TYPE "LBP_typeAxisX"
TITLE = Axis interface / Interfaz de eje / Achsschnittstelle
// User data type for blocks LBP_Axis1 [DB31] .. LBP_Axis31 [DB61] / Tipo de dato de usuario para bloques LBP_Axis1 [DB31] .. LBP_Axis31 [DB61] / Anwender-Datentyp für Bausteine LBP_Axis1 [DB31] .. LBP_Axis31 [DB61]
// stored: IsFailsafeCompliant false
   STRUCT
      A_FD_OR : Byte;   // Vorschub-Override / Feedrate override / Corrección de avance
      A_DriveEnable : Bool;   // Antriebstest-Bewegung aktivieren / Drive test movement enable / Habilitar movimiento test accionamiento
      A_AckFixedStop : Bool;   // Quittieren Festanschlag erreicht / Acknowledge fixed stop reached / Confirmar tope fijo alcanzado
      A_SensorFixedStop : Bool;   // Sensor Festanschlag / Sensor fixed stop / Sensor tope fijo
      A_ASpDisable : Bool;   // Achse/Spindel deaktivieren / Axis/spindle disable / Deshabilitar eje/cabezal
      A_Follow_upMode : Bool;   // Nachlaufbetrieb / Follow-up mode / Modo de seguimiento
      A_PosMeas1 : Bool;   // Positionsmesssystem 1 / Position measuring system 1 / Sistema de medida de posición 1
      A_PosMeas2 : Bool;   // Positionsmesssystem 2 / Position measuring system 2 / Sistema de medida de posición 2
      A_ORactive : Bool;   // Override aktiv / Override active / Corrección activa
      A_SWCam : Bool;   // SW Nocken-Aktivierung / SW cam activation / Activación de levas de SW
      A_ContrEnable : Bool;   // Steuerung aktivieren / Controller enable / Habilitar controlador
      A_DelDTGSpReset : Bool;   // Restweg löschen/Spindel-Reset / Delete distance to go/Spindle-Reset / Borrar trayecto residual/reset de cabezal
      A_Clamp : Bool;   // Spannen läuft / Clamping in progress / Amarre en curso
      A_RefVal1 : Bool;   // Referenzpunktwert 1 / Reference point value 1 / Valor de punto de referencia 1
      A_RefVal2 : Bool;   // Referenzpunktwert 2 / Reference point value 2 / Valor de punto de referencia 2
      A_RefVal3 : Bool;   // Referenzpunktwert 3 / Reference point value 3 / Valor de punto de referencia 3
      A_RefVal4 : Bool;   // Referenzpunktwert 4 / Reference point value 4 / Valor de punto de referencia 4
      A_ExtZO : Bool;   // Externe ZO importieren / Import external ZO / Importar ZO externo
      A_EnabTravFixedStop : Bool;   // Verfahren zu Festanschlag aktivieren / Enable travel to fixed stop / Activar desplazamiento a tope fijo
      A_FixedFD1 : Bool;   // Festen Vorschub 1 aktivieren / Activate fixed feedrate 1 / Activar avance fijo 1
      A_FixedFD2 : Bool;   // Festen Vorschub 2 aktivieren / Activate fixed feedrate 2 / Activar avance fijo 2
      A_FixedFD3 : Bool;   // Festen Vorschub 3 aktivieren / Activate fixed feedrate 3 / Activar avance fijo 3
      A_FixedFD4 : Bool;   // Festen Vorschub 4 aktivieren / Activate fixed feedrate 4 / Activar avance fijo 4
      A_VelocSpeedLimit : Bool;   // Begrenzung Geschwindigkeit/Spindeldrehzahl / Velocity/spindle speed limitation / Limitación velocidad/velocidad de giro cabezal
      A_PrgtestAxRel : Bool;   // Programmtest Achse/Spindel freigeben / Program test axis/spindle release / Habilitar test de programa eje/cabezal
      A_HW1 : Bool;   // Handrad 1 aktivieren / Activate handwheel 1 / Activar volante 1
      A_HW2 : Bool;   // Handrad 2 aktivieren / Activate handwheel 2 / Activar volante 2
      A_HW3 : Bool;   // Handrad 3 aktivieren / Activate handwheel 3 / Activar volante 3
      A_FDSpStop : Bool;   // Vorschub-Stopp/Spindel-Stopp / Feed stop/spindle stop / Parada de avance/parada de cabezal
      A_Disable : Bool;   // Verfahrtaste deaktivieren / Traversing key disable / Desactivar tecla de desplazamiento
      A_RapidTrOR : Bool;   // Eilgang Override / Rapid traverse override / Corregir rápido
      A_Minus : Bool;   // Verfahrtaste minus / Traversing key minus / Tecla desplazamiento Menos
      A_Plus : Bool;   // Verfahrtaste plus / Traversing key plus / Tecla desplazamiento Más
      A_INC1 : Bool;   // INC1
      A_INC10 : Bool;   // INC10
      A_INC100 : Bool;   // INC100
      A_INC1000 : Bool;   // INC1000
      A_INC10000 : Bool;   // INC10000
      A_INCVar : Bool;   // INC-Variable / INC variable / Variable INC
      A_ContManTravel : Bool;   // Kontinuierliches Verfahren von Hand / Continuous manual travel / Desplazamiento continuo a mano
      f5_7 : Bool;
      A_OEMAxis : Byte;   // OEM Achsen-Signale / OEM axis signals / Señales ejes OEM
      A_InvHWDirOfRot : Bool;   // Drehrichtung Handrad umkehren / Inverting handwheel direction of rotation / Invertir sentido de giro volante
      f7_1 : Bool;
      f7_2 : Bool;
      f7_3 : Bool;
      f7_4 : Bool;
      f7_5 : Bool;
      f7_6 : Bool;
      f7_7 : Bool;
      A_NCASpChanA : Bool;   // NC-Achse/Spindel Kanal A zuweisen / Assign NC axis/spindle channel A / Asignar eje/cabezal CN canal A
      A_NCASpChanB : Bool;   // NC-Achse/Spindel Kanal B zuweisen / Assign NC axis/spindle channel B / Asignar eje/cabezal CN canal B
      A_NCASpChanC : Bool;   // NC-Achse/Spindel Kanal C zuweisen / Assign NC axis/spindle channel C / Asignar eje/cabezal CN canal C
      A_NCASpChanD : Bool;   // NC-Achse/Spindel Kanal D zuweisen / Assign NC axis/spindle channel D / Asignar eje/cabezal CN canal D
      A_NCASpStrobe : Bool;   // Activierung der Zuweisung mit pos. Flanke / Activation of assignment with pos. edge / Activación de asignación con flanco pos.
      f8_5 : Bool;
      f8_6 : Bool;
      A_PLCASp : Bool;   // PLC Achse/Spindel anfordern / Request PLC axis/spindle / Solicitar eje/cabezal PLC
      A_Para_A : Bool;   // Regler-Parametersatz Servo A / Parameter block servo A / Bloque de parámetros servo A
      A_Para_B : Bool;   // Regler-Parametersatz Servo B / Parameter block servo B / Bloque de parámetros servo B
      A_Para_C : Bool;   // Regler-Parametersatz Servo C / Parameter block servo C / Bloque de parámetros servo C
      A_LockParSetDef : Bool;   // Parametersatz-Definition aus NC sperren / Lock parameter set definition from NC / Bloquear definición de juego de parámetros desde CN
      f9_4 : Bool;
      f9_5 : Bool;
      f9_6 : Bool;
      f9_7 : Bool;
      A_REPOSDelay : Bool;   // REPOS DELAY
      f10_1 : Bool;
      f10_2 : Bool;
      f10_3 : Bool;
      f10_4 : Bool;
      f10_5 : Bool;
      f10_6 : Bool;
      f10_7 : Bool;
      A_StartBrakeTest : Bool;   // Bremstest starten / Start brake test / Iniciar test de frenado
      f11_1 : Bool;
      f11_2 : Bool;
      f11_3 : Bool;
      f11_4 : Bool;
      f11_5 : Bool;
      f11_6 : Bool;
      f11_7 : Bool;
      A_HWLimitMinus : Bool;   // Hardware-Endschalter minus / Hardware limit switch minus / Final de carrera hardware Menos
      A_HWLimitPlus : Bool;   // Hardware-Endschalter plus / Hardware limit switch plus / Final de carrera hardware Más
      A_SWLimit2Minus : Bool;   // 2. Software-Endschalter minus / 2nd software limit switch minus / 2.º final de carrera software Menos
      A_SWLimit2Plus : Bool;   // 2. Software-Endschalter plus / 2nd software limit switch plus / 2.º final de carrera software Más
      A_ModuloLimitEn : Bool;   // Modulo-Grenze aktiviert / Modulo limit enabled / Límite de módulo habilitado
      f12_5 : Bool;
      f12_6 : Bool;
      A_DelayRef : Bool;   // Referenzpunkt anfahren verzögern / Delay reference point approach / Retardar búsqueda del punto de referencia
      A_JogFixPPos0 : Bool;   // JogFixPointPos 0
      A_JogFixPPos1 : Bool;   // JogFixPointPos 1
      A_JogFixPPos2 : Bool;   // JogFixPointPos 2
      A_JogToPos : Bool;   // Tippbetrieb zu Position / Jog to position / Modo JOG a posición
      f13_4 : Bool;
      f13_5 : Bool;
      f13_6 : Bool;
      f13_7 : Bool;
      A_ProgtestSuppress : Bool;   // Programmtest unterdrücken / Program test to suppress / Suprimir test de programa
      A_ProgtestActivate : Bool;   // Programmtest aktivieren / Activate program test / Activar test de programa
      f14_2 : Bool;
      f14_3 : Bool;
      f14_4 : Bool;
      f14_5 : Bool;
      f14_6 : Bool;
      f14_7 : Bool;
      f15 : Byte;
      A_ActGearA : Bool;   // Aktuelle Getriebestufe A / Actual gear stage A / Escalón de reducción actual A
      A_ActGearB : Bool;   // Aktuelle Getriebestufe B / Actual gear stage B / Escalón de reducción actual B
      A_ActGearC : Bool;   // Aktuelle Getriebestufe C / Actual gear stage C / Escalón de reducción actual C
      A_GearChangeOv : Bool;   // Getriebe hat umgeschaltet / Gear has changed over / El accionamiento ha conmutado
      A_Sp1Syn : Bool;   // Spindel 1 neu synchronisieren / Re-synchronize spindle 1 / Volver a sincronizar cabezal 1
      A_Sp2Syn : Bool;   // Spindel 2 neu synchronisieren / Re-synchronize spindle 2 / Volver a sincronizar cabezal 2
      A_NoMonitorGear : Bool;   // Keine Überwachung bei Getriebeumschaltung / No monitoring when changing gear / Sin vigilancia con cambio de reducción
      A_DeleteS : Bool;   // S-Wert löschen / Delete S value / Borrar valor S
      A_FD_ORSp : Bool;   // Vorschub-Override für Spindel gültig / Feedrate override for spindle valid / Corrección de avance válida para cabezal
      f17_1 : Bool;
      f17_2 : Bool;
      f17_3 : Bool;
      A_Sp1SynP : Bool;   // Spindel 1 für Positionierung neu synchronisieren / Re-synchronize spindle 1 for positioning / Volver a sincronizar cabezal 1 para posicionamiento
      A_Sp2SynP : Bool;   // Spindel 2 für Positionierung neu synchronisieren / Re-synchronize spindle 2 for positioning / Volver a sincronizar cabezal 2 para posicionamiento
      A_M3M4Inv : Bool;   // Invertieren M3/M4 / Invert M3/M4 / Invertir M3/M4
      f17_7 : Bool;
      f18_0 : Bool;
      f18_1 : Bool;
      f18_2 : Bool;
      f18_3 : Bool;
      A_OscilPLC : Bool;   // Pendelbetrieb über PLC / Oscillation via PLC / Oscilación a través de PLC
      A_OscilSpeed : Bool;   // Pendelbetrieb aktivieren / Enable Oscillation / Habilitar oscilación
      A_SetRotDirectRight : Bool;   // Sollwert Schwingrichtung rechts / Setpoint osci. direct. right / Consigna sentido oscilación derecha
      A_SetRotDirectLeft : Bool;   // Sollwert Schwingrichtung links / Setpoint osci. direct. left / Consigna sentido oscilación izquierda
      A_SpOR : Byte;   // Spindel Override / Spindle override / Corrección cabezal
      f20_0 : Bool;
      A_RUEncQuStop : Bool;   // Hochlaufgeber Schnellstopp / Run-up encoder quick stop / Parada rápida generador de rampa
      f20_2 : Bool;
      A_SpeedSetpSmooth : Bool;   // Drehzahlsollwert-Glättung / Speed setpoint smoothing / Alisado consigna velocidad de giro
      f20_4 : Bool;
      A_HoldBrakeToOpen : Bool;   // Haltebremse offen / Holding brake open / Freno de mantenimiento abierto
      f20_6 : Bool;
      f20_7 : Bool;
      A_ParA : Bool;   // Parametersatz-Auswahl A / Parameter set selection A / Selección juego de parámetros A
      A_ParB : Bool;   // Parametersatz-Auswahl B / Parameter set selection B / Selección juego de parámetros B
      A_ParC : Bool;   // Parametersatz-Auswahl C / Parameter set selection C / Selección juego de parámetros C
      A_MotA : Bool;   // Auswahl Motor A / Motor selection A / Selección motor A
      A_MotB : Bool;   // Auswahl Motor B / Motor selection B / Selección motor B
      A_MotOK : Bool;   // Motor ausgewählt / Motor selected / Motor seleccionado
      A_IntegratDisable : Bool;   // N-Steuerung Integrator deaktivieren / N controller integrator disable / Desactivar controlador N integrador
      A_PulseEnable : Bool;   // Impuls aktivieren / Pulse enable / Habilitar impulsos
      f22_0 : Bool;
      f22_1 : Bool;
      f22_2 : Bool;
      f22_3 : Bool;
      f22_4 : Bool;
      f22_5 : Bool;
      f22_6 : Bool;
      f22_7 : Bool;
      f23_0 : Bool;
      f23_1 : Bool;
      f23_2 : Bool;
      f23_3 : Bool;
      f23_4 : Bool;
      f23_5 : Bool;
      f23_6 : Bool;
      f23_7 : Bool;
      A_RotationMonit : Bool;   // Schrittmotor: Drehüberwachung / Stepper motor: Rotation monitoring / Motor paso a paso: vigilancia de velocidad
      A_ControlAx : Bool;   // Steuerungsachse / Control Axis / Eje de control
      f24_2 : Bool;
      f24_3 : Bool;
      A_TorqComp : Bool;   // Drehmoment-Kompensation / Torque compensation / Compensación de par
      A_ChangSetpOutAss0 : Bool;   // Bitwert für CTRLOUT_changed - Sollwertausgang-Zuordnung ändern / Bit value for CTRLOUT_changed - Change setpoint output assignment / Valor de bit para CTRLOUT_changed - Modificar asignación de salida de consigna
      A_ChangSetpOutAss1 : Bool;   // Bitwert für CTRLOUT_changed - Sollwertausgang-Zuordnung ändern / Bit value for CTRLOUT_changed - Change setpoint output assignment / Valor de bit para CTRLOUT_changed - Modificar asignación de salida de consigna
      A_MS : Bool;   // Master / Slave Ein / Master / Slave On / Maestro/esclavo Con
      A_DynBComp : Bool;   // Dynamische Spielkompensation aktiviert / Dynamic backlash compensation activated / Compensación dinámica de juego activada
      f25_1 : Bool;
      f25_2 : Bool;
      f25_3 : Bool;
      f25_4 : Bool;
      f25_5 : Bool;
      f25_6 : Bool;
      f25_7 : Bool;
      f26_0 : Bool;
      f26_1 : Bool;
      f26_2 : Bool;
      A_CompContr : Bool;   // Kompensation Steuerung Ein / Compensation controller On / Compensación controlador Con
      A_FollowAxOv : Bool;   // Override Folgeachse aktivieren / Enable following axis override / Habilitar corrección eje esclavo
      f26_5 : Bool;
      f26_6 : Bool;
      f26_7 : Bool;
      A_DEPMCS : Bool;   // Fortsetzen: DEPMCS / Resume: DEPMCS / Continuar: DEPMCS
      A_DEPBCS : Bool;   // Fortsetzen: DEPBCS / Resume: DEPBCS / Continuar: DEPBCS
      A_Corr : Bool;   // Fortsetzen: Korr / Resume: Corr / Continuar: corr
      A_HIAxMove : Bool;   // Fortsetzen: HIAxMove / Resume: HIAxMove / Continuar: HIAxMove
      A_StopDEPMCS : Bool;   // Stopp: DEPMCS / Stop: DEPMCS / Parada: DEPMCS
      A_StopDEPBCS : Bool;   // Stopp: DEPBCS / Stop: DEPBCS / Parada: DEPBCS
      A_StopCorr : Bool;   // Stopp: Korr / Stop: Corr / Parada: corr
      A_StopHIAxMove : Bool;   // Stopp: HIAxMove / Stop: HIAxMove / Parada: HIAxMove
      A_OscillAxExtRev : Bool;   // OscillAxExtReversal
      A_AxReset : Bool;   // AXRESET
      A_AxResume : Bool;   // AXRESUME
      A_SetRP : Bool;   // Umkehrpunkt setzen / Set reversal point / Definir punto de inversión
      A_ChangeRP : Bool;   // Umkehrpunkt ändern / Change reversal point / Cambiar punto de inversión
      A_StopRP : Bool;   // Stopp am nächsten Umkehrpunkt / Stop at next reversal point / Parar en siguiente punto de inversión
      A_Stop : Bool;   // Stopp / Stop / Parada
      A_PLCAxis : Bool;   // PLC prüft Achse / PLC checks axis / PLC comprueba eje
      f29_0 : Bool;
      f29_1 : Bool;
      f29_2 : Bool;
      f29_3 : Bool;
      A_StartGantSynRun : Bool;   // Portal-Synchronisationslauf starten / Start gantry synchronization run / Iniciar sincronización Gantry
      A_NoAutoSync : Bool;   // Kein Auto Sync / No auto sync / Sin sinc auto
      f29_6 : Bool;
      f29_7 : Bool;
      A_StopSpindle : Bool;   // Spindel stoppen / Stop spindle / Parar cabezal
      A_StartCW : Bool;   // Spindel rechtsdrehend starten / Start spindle clockwise / Iniciar cabezal con giro a derecha
      A_StartCCW : Bool;   // Spindel linksdrehend starten / Start spindle counterclockwise / Iniciar cabezal con giro a izquierda
      A_AutoGearStep : Bool;   // Autom. Getriebestufen-Änderung / Autom. gear step change / Cambio automático de escalón de reducción
      A_PosSpindle : Bool;   // Spindel positionieren / Position spindle / Posicionar cabezal
      f30_5 : Bool;
      f30_6 : Bool;
      f30_7 : Bool;
      f31_0 : Bool;
      f31_1 : Bool;
      f31_2 : Bool;
      f31_3 : Bool;
      A_Resynchronize : Bool;   // Neu synchronisieren / Resynchronize / Volver a sincronizar
      A_DisSync : Bool;   // Synchronisation deaktivieren / Disable synchronization / Desactivar sincronización
      A_Tracksync : Bool;   // Synchronlauf verfolgen / Track synchronism / Seguir marcha síncrona
      A_DelSyncRunCorr : Bool;   // Löschen synchrone Laufkorrektur / Deleting synchronous run correction / Borrar corrección de sincronismo
      f32_0 : Bool;
      f32_1 : Bool;
      f32_2 : Bool;
      f32_3 : Bool;
      f32_4 : Bool;
      f32_5 : Bool;
      f32_6 : Bool;
      f32_7 : Bool;
      f33_0 : Bool;
      f33_1 : Bool;
      f33_2 : Bool;
      f33_3 : Bool;
      f33_4 : Bool;
      f33_5 : Bool;
      f33_6 : Bool;
      f33_7 : Bool;
      A_SI_SetpLimBit0 : Bool;   // Sollwertbegrenzung Bit 0 / Set point limitation Bit0 / Limitación de consigna Bit 0
      A_SI_SetpLimBit1 : Bool;   // Sollwertbegrenzung Bit 1 / Set point limitation Bit1 / Limitación de consigna Bit 1
      f34_2 : Bool;
      f34_3 : Bool;
      f34_4 : Bool;
      f34_5 : Bool;
      f34_6 : Bool;
      f34_7 : Bool;
      f35 : Byte;
      f36 : Array[36..55] of Byte;
      A_FeedDriveCAxEng : Bool;   // Separater Vorschubantrieb als C-Achse eingeschaltet / Separate feed drive as C axis engaged / Accionamiento de avance separado conectado como eje C
      A_SpSpeedDisp : Bool;   // Spindeldrehzahl-Anzeige / Spindle speed display / Indicador velocidad giro cabezal
      A_SpInsideClamp : Bool;   // Spindel-Innenspannen / Spindle inside clamping / Amarre interno cabezal
      f56_3 : Bool;
      f56_4 : Bool;
      f56_5 : Bool;
      f56_6 : Bool;
      f56_7 : Bool;
      f57 : Byte;
      f58 : Word;
      E_SpNA : Bool;   // Spindel/keine Achse / Spindle/no axis / Cabezal/no hay eje
      E_NCU_Link : Bool;   // NCU_link aktive Achse / NCU_link active axis / Eje activo NCU_link
      E_EncodFreq1 : Bool;   // Geber-Grenzfrequenz 1 überschritten / Encoder limit frequency 1 exceeded / Frecuencia límite encóder 1 rebasada
      E_EncodFreq2 : Bool;   // Geber-Grenzfrequenz 2 überschritten / Encoder limit frequency 2 exceeded / Frecuencia límite encóder 2 rebasada
      E_RefSyn1 : Bool;   // Referenziert/synchronisiert 1 / Referenced/synchronized 1 / Referenciado/sincronizado 1
      E_RefSyn2 : Bool;   // Referenziert/synchronisiert 2 / Referenced/synchronized 2 / Referenciado/sincronizado 2
      E_ExactCoarse : Bool;   // Position erreicht mit exaktem Stopp grob / Position reached with exact stop coarse / Posición alcanzada con parada exacta gruesa
      E_ExactFine : Bool;   // Position erreicht mit exaktem Stopp fein / Position reached with exact stop fine / Posición alcanzada con parada exacta fina
      E_TravRequ : Bool;   // Verfahranforderung / Travel request / Solicitud desplazamiento
      E_AxialAlarm : Bool;   // Achsen-Alarm / Axial alarm / Alarma axial
      E_AxisReady : Bool;   // Achse bereit / Axis ready / Eje listo
      E_Follow_upMode : Bool;   // Folgemodus aktiv / Follow-up mode active / Modo de seguimiento activo
      E_Stat : Bool;   // Achse/Spindel im Stillstand (n<nmin) / Axis/spindle stationary (n<nmin) / Eje/cabezal en parada (n<nmin)
      E_PositContr : Bool;   // Positionssteuerung aktiv / Position controller active / Control de posición activo
      E_SpeedContr : Bool;   // Drehzahlregler aktiv / Speed controller active / Regulador de velocidad activo
      E_CurrentContr : Bool;   // Aktuelle Steuerung aktiv / Current controller active / Controlador actual activo
      E_SWCam : Bool;   // Software-Nocken aktiv / Software cams active / Levas de software activas
      E_HWOverlay : Bool;   // Handrad-Overlay aktiv / Handwheel overlay active / Overlay volante activo
      E_RevFD : Bool;   // Umdrehungsvorschub aktiv / Revolutional feedrate active / Avance revoluciones activo
      E_MeasAct : Bool;   // Messung aktiv / Measuring active / Medición activa
      E_ActTravFStop : Bool;   // Verfahren zu Festanschlag aktivieren / Enable travel to fixed stop / Activar desplazamiento a tope fijo
      E_FixedStop : Bool;   // Festanschlag erreicht / Fixed stop reached / Tope fijo alcanzado
      E_ForceFixedStop : Bool;   // Kraft Festanschlag begrenzt / Force fixed stop limited / Fuerza tope fijo limitada
      E_AxContainerRot : Bool;   // Achscontainer Drehung aktiv / Axis container rotation active / Giro contenedor de ejes activo
      E_AxReset : Bool;   // Achsen-Reset durchgeführt / Axis reset done / Reset ejes realizado
      E_PLCCtrlAx : Bool;   // PLC gesteuerte Achse / PLC controlled axis / Eje controlado por PLC
      E_AxStop : Bool;   // Achsen-Stopp aktiv / Axis stop active / Parada de ejes activa
      E_AxSpDisable : Bool;   // Deaktivierung Achse/Spindel aktiv / Axis/spindle disable active / Desactivación eje/cabezal activa
      E_StopDEPMCS : Bool;   // Stopp DEPMCS aktiv / Stop DEPMCS active / Detener DEPMCS activo
      E_StopDEPBCS : Bool;   // Stopp DEPBCS aktiv / Stop DEPBCS active / Detener DEPBCS activo
      E_StopCorr : Bool;   // Stopp Korr aktiv / Stop Corr active / Detener corr activo
      E_StopHIAxMove : Bool;   // Stopp HIAxMove aktiv / Stop HIAxMove active / Detener HIAxMove activo
      E_HW1 : Bool;   // Handrad 1 aktiv / Handwheel 1 active / Volante 1 activo
      E_HW2 : Bool;   // Handrad 2 aktiv / Handwheel 2 active / Volante 2 activo
      E_HW3 : Bool;   // Handrad 3 aktiv / Handwheel 3 active / Volante 3 activo
      f64_3 : Bool;
      E_TReqMinus : Bool;   // Verfahranforderung minus / Travel request minus / Solicitud desplazamiento Menos
      E_TReqPlus : Bool;   // Verfahranforderung plus / Travel request plus / Solicitud desplazamiento Más
      E_TCMinus : Bool;   // Verfahrbefehl minus / Traverse command minus / Comando de desplazamiento Menos
      E_TCPlus : Bool;   // Verfahrbefehl plus / Traverse command plus / Comando de desplazamiento Más
      E_INC1 : Bool;   // INC1
      E_INC10 : Bool;   // INC10
      E_INC100 : Bool;   // INC100
      E_INC1000 : Bool;   // INC1000
      E_INC10000 : Bool;   // INC10000
      E_INCVar : Bool;   // INC-Variable / INC variable / Variable INC
      E_ContManTravelAct : Bool;   // Kontinuierliches manuelles Verfahren aktiv / Continuous manual travel active / Desplazamiento manual continuo activo
      f65_7 : Bool;
      E_OEMAxis : Byte;   // OEM Achsen-Signale / OEM axis signals / Señales ejes OEM
      E_InvHWDirOfRot : Bool;   // Handrad-Drehrichtung invertiert aktiv / Handwheel direction of rotation invert actively / Invertir activamente sentido de giro volante
      f67_1 : Bool;
      f67_2 : Bool;
      f67_3 : Bool;
      f67_4 : Bool;
      f67_5 : Bool;
      f67_6 : Bool;
      f67_7 : Bool;
      E_NCASpChanA : Bool;   // NC Achse/Spindel in Kanal A / NC axis/spindle in channel A / Eje/cabezal CN en canal A
      E_NCASpChanB : Bool;   // NC Achse/Spindel in Kanal B / NC axis/spindle in channel B / Eje/cabezal CN en canal B
      E_NCASpChanC : Bool;   // NC Achse/Spindel in Kanal C / NC axis/spindle in channel C / Eje/cabezal CN en canal C
      E_NCASpChanD : Bool;   // NC Achse/Spindel in Kanal D / NC axis/spindle in channel D / Eje/cabezal CN en canal D
      E_PLCType : Bool;   // Neuer Typ von PLC angefordert / New type requested by PLC / Nuevo tipo solicitado por PLC
      E_ChPoss : Bool;   // Achse ändern möglich / Change axis possible / Cambio de eje posible
      E_NeutrASp : Bool;   // Neutrale Achse/Spindel / Neutral axis/spindle / Eje/cabezal neutro
      E_PLCASp : Bool;   // PLC Achse/Spindel / PLC axis/spindle / Eje/cabezal PLC
      E_ParS_A : Bool;   // Regler-Parametersatz Servo A / Parameter block servo A / Bloque de parámetros servo A
      E_ParS_B : Bool;   // Regler-Parametersatz Servo B / Parameter block servo B / Bloque de parámetros servo B
      E_ParS_C : Bool;   // Regler-Parametersatz Servo C / Parameter block servo C / Bloque de parámetros servo C
      E_NCUNumLink_3 : Bool;
      E_NCUNumLink_4 : Bool;
      E_NCUNumLink_5 : Bool;
      E_NCUNumLink_6 : Bool;
      E_NCUNumLink_7 : Bool;
      E_ReposSh : Bool;   // REPOS Verschiebung / REPOS shift / Decalaje REPOS
      E_ReposShValid : Bool;   // REPOS Verschiebung gültig / REPOS shift valid / Decalaje REPOS válido
      E_ReposDelayQuit : Bool;   // REPOS Verzögerung beenden / REPOS delay quit / Finalizar retardo REPOS
      f70_3 : Bool;
      f70_4 : Bool;
      E_SI_Drv_SICSCC : Bool;   // DRV-Safety Integrated mit SIC/SCC aktiv / DRV-Safety Integrated with SIC/SCC active / DRV Safety Integrated con SIC/SCC activo
      f70_6 : Bool;
      f70_7 : Bool;
      E_BrakeTest : Bool;   // Bremstest aktiv / Brake test active / Test de frenado activo
      f71_1 : Bool;
      f71_2 : Bool;
      f71_3 : Bool;
      E_POS_RESTORED1 : Bool;   // POS_RESTORED 1
      E_POS_RESTORED2 : Bool;   // POS_RESTORED 2
      f71_6 : Bool;
      E_PLCAxDedic : Bool;   // PLC Achse dediziert / PLC axis dedicated / Eje PLC dedicado
      E_MMC_REPOSDelay : Bool;   // HMI REPOS DELAY
      f72_1 : Bool;
      f72_2 : Bool;
      f72_3 : Bool;
      f72_4 : Bool;
      f72_5 : Bool;
      f72_6 : Bool;
      f72_7 : Bool;
      f73 : Byte;
      f74_0 : Bool;
      f74_1 : Bool;
      f74_2 : Bool;
      f74_3 : Bool;
      E_ModLimEnAct : Bool;   // Modulo-Grenze aktiviert aktiv / Modulo limit enabled active / Límite de módulo habilitado activo
      f74_5 : Bool;
      f74_6 : Bool;
      f74_7 : Bool;
      E_JogFixPPos0Act : Bool;   // JogFixPointPos 0 aktiv / JogFixPointPos 0 active / JogFixPointPos 0 activo
      E_JogFixPPos1Act : Bool;   // JogFixPointPos 1 aktiv / JogFixPointPos 1 active / JogFixPointPos 1 activo
      E_JogFixPPos2Act : Bool;   // JogFixPointPos 2 aktiv / JogFixPointPos 2 active / JogFixPointPos 2 activo
      E_JogFixPPos0 : Bool;   // JogFixPointPos 0 erreicht / JogFixPointPos 0 reached / JogFixPointPos 0 alcanzado
      E_JogFixPPos1 : Bool;   // JogFixPointPos 1 erreicht / JogFixPointPos 1 reached / JogFixPointPos 1 alcanzado
      E_JogFixPPos2 : Bool;   // JogFixPointPos 2 erreicht / JogFixPointPos 2 reached / JogFixPointPos 2 alcanzado
      E_JogToPos : Bool;   // Tippbetrieb zu Position aktiv / Jog to position active / Modo JOG a posición activo
      E_JogPos : Bool;   // Jog-Position erreicht / Jog position reached / Posición JOG alcanzada
      E_ScratchPulse : Bool;   // Scratch Impuls / Scratch pulse / Impulso de aproximación con contacto
      f76_1 : Bool;
      f76_2 : Bool;
      f76_3 : Bool;
      E_PathAxis : Bool;   // Bahnachse / Path axis / Eje de trayectoria
      E_PosAxis : Bool;   // Positionierungsachse / Positioning axis / Eje de posicionamiento
      E_IndexAxisPos : Bool;   // Indexachse in Position / Indexing axis in position / Eje de indexado en posición
      E_CurvePos : Bool;   // Kurvenachse in Position / Curve axis in position / Eje de leva en posición
      E_CollCheckRedSpeed : Bool;   // Reduzierte Geschwindigkeit der Kollisionsprüfung / Reduced speed of Collisions Check / Velocidad de comprobación de colisiones reducida
      f77_1 : Bool;
      f77_2 : Bool;
      f77_3 : Bool;
      f77_4 : Bool;
      f77_5 : Bool;
      f77_6 : Bool;
      f77_7 : Bool;
      E_FPosAxis : Real;   // F-Funktion (REAL-Format) für Positionierungsachsen / F function (REAL format) for positioning axes / Función F (formato REAL) para ejes de posicionamiento
      E_SetpGearA : Bool;   // Sollwert-Getriebestufe A / Setpoint gear stage A / Consigna de escalón de reducción A
      E_SetpGearB : Bool;   // Sollwert-Getriebestufe B / Setpoint gear stage B / Consigna de escalón de reducción B
      E_SetpGearC : Bool;   // Sollwert-Getriebestufe C / Setpoint gear stage C / Consigna de escalón de reducción C
      E_GearChange : Bool;   // Getriebe-Umschaltung / Gear changeover / Cambio de reducción
      f82_4 : Bool;
      f82_5 : Bool;
      f82_6 : Bool;
      f82_7 : Bool;
      E_SpeedLimit : Bool;   // Drehzahlgrenzwert überschritten / Speed limit exceeded / Límite de velocidad rebasado
      E_SetSpeedLimit : Bool;   // Solldrehzahl begrenzt / Setpoint speed limited / Velocidad de cabezal limitada
      E_SetSpeedIncreased : Bool;   // Solldrehzahl erhöht / Setpoint speed increased / Velocidad de cabezal aumentada
      E_GeoMonit : Bool;   // Geometrie-Überwachung / Geometry monitoring / Vigilancia de geometría
      E_SupportAreaViol : Bool;   // Auflage Bereichsgrenzen verletzt / Support area limits violated / Límites zona de admisión vulnerados
      E_SetRange : Bool;   // Spindel im Sollbereich / Spindle in setpoint range / Cabezal en rango de consigna
      E_SpeedMonit : Bool;   // Drehzahlüberwachung / Speed monitoring / Vigilancia de velocidad
      E_ActRotRight : Bool;   // Istdrehrichtung rechts / Actual rotation direction right / Sentido de giro actual derecha
      E_ConstCuttSpeed : Bool;   // Konst. Schnittgeschwindigkeit aktiv / Const. cutting speed active / Velocidad de corte const. activa
      E_SUG : Bool;   // SUG aktiv (Drehzahl der Schleifscheiben-Oberfläche) / SUG active (grinding wheel surface speed) / SUG activo (velocidad de giro de la superficie de la muela de refrentar)
      E_CLG : Bool;   // CLG aktiv / CLG active / CLG activo
      E_Tapping : Bool;   // Gewindebohren ohne Ausgleichsfutter / Tapping without compensating chuck / Roscado sin mandril de compensación
      E_SyncMode : Bool;   // Synchronbetrieb Spindel aktiv / Synchronous mode spindle active / Modo de sincronización cabezal activo
      E_PosMode : Bool;   // Positionsbetrieb Spindel aktiv / Positioning mode spindle active / Modo de posicionamiento cabezal activo
      E_OscillMode : Bool;   // Pendelbetrieb Spindel aktiv / Oscillation mode spindle active / Modo de oscilación cabezal activo
      E_ContrMode : Bool;   // Steuermodus Spindel aktiv / Control mode spindle active / Modo de control cabezal activo
      E_ToolDynLimit : Bool;   // Werkzeug mit dynamischer Grenze / Tool with dynamics limit / Herramienta con límite dinámico
      f85_1 : Bool;
      f85_2 : Bool;
      f85_3 : Bool;
      f85_4 : Bool;
      E_SpInPosition : Bool;   // Spindel in Position / Spindle in position / Cabezal en posición
      f85_6 : Bool;
      f85_7 : Bool;
      E_MFunct : Int;   // M-Funktion (INT) für Spindel / M function (INT) for spindle / Función M (INT) para cabezal
      E_SFunct : Real;   // S-Function (REAL) für Spindel / S function (REAL) for spindle / Función S (REAL) para cabezal
      f92_0 : Bool;
      E_RUEncDisabl : Bool;   // Hochlaufgeber-Sperre aktiv / Run-up encoder disable active / Deshabilitación generador de rampa activa
      f92_2 : Bool;
      E_SpeedSetpSmooth : Bool;   // Drehzahlsollwert Glättung aktiv / Speed setpoint smoothing active / Alisado de consigna de velocidad activo
      E_RLIact : Bool;   // RLI aktiv / RLI active / RLI activo
      E_HoldBrakeOpened : Bool;   // Haltebremse geöffnet / Holding brake opened / Freno de mantenimiento abierto
      f92_6 : Bool;
      E_DriveRunEn : Bool;   // Antriebslauf aktiviert / Drive run enabled / Marcha de accionamiento habilitada
      E_ParA : Bool;   // Aktiver Parametersatz A / Active parameter set A / Juego de parámetros A activo
      E_ParB : Bool;   // Aktiver Parametersatz B / Active parameter set B / Juego de parámetros B activo
      E_ParC : Bool;   // Aktiver Parametersatz C / Active parameter set C / Juego de parámetros C activo
      E_MotA : Bool;   // Aktiver Motor A / Active motor A / Motor activo A
      E_MotB : Bool;   // Aktiver Motor B / Active motor B / Motor activo B
      E_MotOK : Bool;   // Antrieb bereit / Drive ready / Accionamiento listo
      E_IntegratDisable : Bool;   // N-Steuerung Integrator deaktiviert / N controller integrator disabled / Controlador N integrador desactivado
      E_PulseEnable : Bool;   // Impulse aktiviert / Pulses enabled / Impulsos activados
      E_MTempWarn : Bool;   // Temperaturvorwarnung Motor / Prewarning motor temperature / Prealarma temperatura motor
      E_HTempWarn : Bool;   // Temperaturvorwarnung Kühlkörper / Prewarning heat sink temperature / Prealarma temperatura disipador
      E_RUComplete : Bool;   // Hochlauf abgeschlossen / Ramp-up complete / Arranque finalizado
      E_MdMdx : Bool;   // Md<Mdx
      E_NactNmin : Bool;   // nact<nmin
      E_NactNx : Bool;   // nact<nx
      E_NactNset : Bool;   // nact=nset
      E_Message : Bool;   // Variable Meldungsfunktion 1 / Variable message function 1 / Función de avisos variable 1
      E_UDClessAlThreshold : Bool;   // UDC-Verbindung < Alarmschwelle / UDC-link < alarm threshold / Conexión UDC < umbral de alarma
      E_DcVoltageAlarmAct : Bool;   // ESR: Zwischenkreisspannung liegt unter dem festgelegten Minimum / ESR: DC link voltage is below the specified minimum / ESR: la tensión del circuito intermedio está por debajo del mínimo establecido
      E_GeneratorOperationAct : Bool;   // ESR: Generatorischer Betrieb aktiv / ESR: generator operation is active / ESR: modo generador activo
      E_SpeedBelowMin : Bool;   // ESR: Ist-Drehzahl liegt unter der festgelegten Mindestdrehzahl - Achse ist Generatorachse / ESR: actual speed is below specified minimum speed - axis is a generator axis / ESR: la velocidad real está por debajo de la velocidad mín. establecida - el eje es un eje generador
      E_Message2 : Bool;   // Variable Meldungsfunktion 2 / Variable message function 2 / Función de avisos variable 2
      E_Message3 : Bool;   // Variable Meldungsfunktion 3 / Variable message function 3 / Función de avisos variable 3
      f95_6 : Bool;
      E_I2TLimit : Bool;   // Leistungsteil I2T Grenze / Power Section I2T limit / Etapa de potencia límite I2T
      E_SpindleMonit : Bool;   // Fehler Spindelüberwachung / Error spindle monitoring / Error vigilancia de cabezal
      E_AxisCtrl : Bool;   // Achsensteuerung aktiv / Axis control active / Control de ejes activo
      E_MSFine : Bool;   // Master/Slave fein / Master/Slave fine / Maestro/esclavo fino
      E_MSCoarse : Bool;   // Master/Slave grob / Master/Slave coarse / Maestro/esclavo grueso
      E_MSCompContr : Bool;   // Master/Slave Kompensationssteuerung aktiviert / Master/Slave compensation controller activated / Control de compensación maestro/esclavo activado
      E_BitValCtrlOutChang0 : Bool;   // Bitwert für CTRLOUT_changed 0: Zuordnung Sollwertausgang ändern / Bit value for CTRLOUT_changed 0: Change setpoint output assignment / Valor de bit CTRLOUT_changed 0: modificar asignación de salida de consigna
      E_BitValCtrlOutChang1 : Bool;   // Bitwert für CTRLOUT_changed 1: Zuordnung Sollwertausgang ändern / Bit value for CTRLOUT_changed 1: Change setpoint output assignment / Valor de bit CTRLOUT_changed 1: modificar asignación de salida de consigna
      E_MS : Bool;   // Master/Slave aktiv / Master/Slave active / Maestro/esclavo activo
      f97 : Byte;
      E_SyncronFine : Bool;   // Feinsynchronisierung / Synchronism fine / Sincronización fina
      E_SyncronCoarse : Bool;   // Grobsynchronisierung / Synchronism coarse / Sincronización gruesa
      E_ActValCoupling : Bool;   // Istwert Koppeln / Actual value coupling / Acoplamiento valor real
      f98_3 : Bool;
      E_OverlayMotion : Bool;   // Überlagerte Bewegung / Overlaid motion / Movimiento superpuesto
      E_SWL : Bool;   // Warngrenze für Geschwindigkeit erreicht / Speed warning limit reached / Límite de alarma de velocidad alcanzado
      E_AWL : Bool;   // Warngrenzwert für Beschleunigung erreicht / Acceleration warning limit reached / Límite de alarma de aceleración alcanzado
      E_EmRetr : Bool;   // Notrückzug aktiv / Emergency retraction active / Retirada de emergencia activa
      E_MasterSp : Bool;   // Master-Spindel / Master spindle / Cabezal maestro
      E_SlaveSp : Bool;   // Slave-Spindel / Slave spindle / Cabezal esclavo
      E_SyncRunCorrDOut : Bool;   // Synchronlauf Korrektur ausgelaufen / Synchronous run correction driven out / Corrección sincronización desviada
      E_AxisAccel : Bool;   // Achse beschleunigt / Axis accelerated / Eje acelera
      E_Sync : Bool;   // Synchronisation aktiv / Synchronization active / Sincronización activa
      E_MSR : Bool;   // Max. Geschwindigkeit erreicht / Max. speed reached / Máx. velocidad alcanzada
      E_MAR : Bool;   // Max. Beschleunigung erreicht / Max. acceleration reached / Máx. aceleración alcanzada
      f99_7 : Bool;
      f100_0 : Bool;
      f100_1 : Bool;
      E_OscillAxExtRev : Bool;   // OscillAxExt Umkehr aktiv / OscillAxExt Reversal active / OscillAxExt inversión activa
      E_StopOscill : Bool;   // Pendelbetrieb kann nicht starten / Oscillation cannot start / No es posible iniciar oscilación
      E_ErrorOscill : Bool;   // Fehler beim Pendeln / Error during oscillation / Error durante oscilación
      E_SparkOut : Bool;   // Ausfeuern aktiv / Spark-out active / Afinado activo
      E_OscillMotion : Bool;   // Pendelbewegung aktiv / Oscillation motion active / Movimiento de oscilación activo
      E_Oscill : Bool;   // Pendelbetrieb aktiv / Oscillation active / Oscilación activa
      f101_0 : Bool;
      f101_1 : Bool;
      E_GantCOLimit : Bool;   // Portal-Abschaltgrenze erreicht / Gantry cut-off limit exceeded / Límite desconexión Gantry alcanzado
      E_GantWarn : Bool;   // Portal-Warngrenze überschritten / Gantry warning limit exceeded / Límite alarma Gantry alcanzado
      E_SynRunStart : Bool;   // Synchronisationslauf startbereit / Synchronization run ready to start / Sincronización lista para iniciar
      E_GantGroupSyn : Bool;   // Portal-Gruppierung ist synchron / Gantry grouping is synchronous / Agrupación Gantry es síncrona
      E_GantLeadAxis : Bool;   // Portal-Führungsachse / Gantry leading axis / Eje maestro Gantry
      E_GantAxis : Bool;   // Portalachse / Gantry axis / Eje Gantry
      E_DynBComp : Bool;   // Dynamische Spielkompensation aktiviert / Dynamic backlash compensation activated / Compensación dinámica de juego activada
      f102_1 : Bool;
      f102_2 : Bool;
      E_ClampTolerance : Bool;   // Spanntoleranz überschritten / Clamp tolerance exceeded / Tolerancia de amarre superada
      f102_4 : Bool;
      E_PosMeas1 : Bool;   // Positionsmesssystem 1 aktiv / Position measuring system 1 active / Sistema de medida de posición 1 activo
      E_PosMeas2 : Bool;   // Positionsmesssystem 2 aktiv / Position measuring system 2 active / Sistema de medida de posición 2 activo
      f102_7 : Bool;
      E_SyncRunCorrIncl : Bool;   // Synchronlauf Korrektur ist eingeschlossen / Synchronous run correction is included / Corrección sincronización incluida
      f103_1 : Bool;
      f103_2 : Bool;
      f103_3 : Bool;
      E_Syncron2Fine : Bool;   // Feinsynchronisierung / Synchronism fine / Sincronización fina
      E_Syncron2Coarse : Bool;   // Grobsynchronisierung / Synchronism coarse / Sincronización gruesa
      f103_6 : Bool;
      f103_7 : Bool;
      E_AIAxis : Array[1..31] of Bool;   // Aktive Zustellachse [1..31] / Active infeed axis[1..31] / Eje de penetración activo [1..31]
      f108_0 : Bool;
      f108_1 : Bool;
      f108_2 : Bool;
      f108_3 : Bool;
      f108_4 : Bool;
      f108_5 : Bool;
      f108_6 : Bool;
      f108_7 : Bool;
      f109_0 : Bool;
      f109_1 : Bool;
      f109_2 : Bool;
      f109_3 : Bool;
      f109_4 : Bool;
      f109_5 : Bool;
      f109_6 : Bool;
      f109_7 : Bool;
      f110_0 : Bool;
      f110_1 : Bool;
      f110_2 : Bool;
      f110_3 : Bool;
      f110_4 : Bool;
      f110_5 : Bool;
      f110_6 : Bool;
      f110_7 : Bool;
      f111_0 : Bool;
      f111_1 : Bool;
      f111_2 : Bool;
      f111_3 : Bool;
      f111_4 : Bool;
      f111_5 : Bool;
      f111_6 : Bool;
      f111_7 : Bool;
      f112 : Byte;
      f113 : Byte;
      f114 : Byte;
      f115 : Byte;
      f116 : Byte;
      f117_0 : Bool;
      f117_1 : Bool;
      f117_2 : Bool;
      f117_3 : Bool;
      f117_4 : Bool;
      f117_5 : Bool;
      f117_6 : Bool;
      f117_7 : Bool;
      f118 : DWord;
      f122 : DWord;
      f126 : Word;   // Intern / Internal / Interno
      E_MMC_ProgtestSuppress : Bool;   // HMI->PLC: Programmtest unterdrücken / HMI->PLC: Suppress program test / HMI->PLC: suprimir test de programa
      E_MMC_ProgtestActivate : Bool;   // HMI->PLC: Programmtest aktivieren / HMI->PLC: Activate program test / HMI->PLC: activar test de programa
      f128_2 : Bool;
      f128_3 : Bool;
      f128_4 : Bool;
      f128_5 : Bool;
      f128_6 : Bool;
      f128_7 : Bool;
      f129 : Byte;
      f130 : Word;
      E_SensorAv : Bool;   // Sensoren verfügbar / Sensors available / Sensores disponibles
      E_S1aMeasARod : Bool;   // Sensor S1: analoge Messposition der Stange / Sensor S1: analogous measurement position of actuating rod / Sensor S1: posición de medida analógica del varillaje
      f132_2 : Bool;
      f132_3 : Bool;
      E_S4dPistonStopP : Bool;   // Sensor S4: Digitalwert Kolben-Stopp-Position / Sensor S4: digital value piston stop position / Sensor S4: valor digital posición de parada del émbolo
      E_S5dAngleShaft : Bool;   // Sensor S5: Digitalwert Winkellage Welle / Sensor S5: digital value angle situation shaft / Sensor S5: valor digital posición angular eje
      E_S6Temp : Bool;   // Sensor S6: Temperatur / Sensor S6: temperature / Sensor S6: temperatura
      f132_7 : Bool;
      f133 : Byte;
      E_ClampingState : Int;   // Zustand des Spannsystems / State of the clamping system / Estado del sistema de amarre
      E_AnalogSensor : Int;   // Analogsensor am Motor / Analog sensor on the motor / Sensor analógico en el motor
      f138_0 : Bool;
      f138_1 : Bool;
      f138_2 : Bool;
      f138_3 : Bool;
      E_S4PistonStopP : Bool;   // Sensor S4: Kolben-Stopp-Position / Sensor S4: piston stop position / Sensor S4: posición de parada del émbolo
      E_S5AngleShaft : Bool;   // Sensor S5: Winkellage Welle / Sensor S5: angle situation shaft / Sensor S5: posición angular eje
      f138_6 : Bool;
      f138_7 : Bool;
      f139 : Byte;
      SCC : Struct   // PLC zu Antrieb (SCC) / PLC to Drive (SCC) / PLC a accionamiento (SCC)
         CW1 : Struct
            TeststopStart : Bool;   // Test-Stopps für erweiterte Funktionen / Test stops for extended functions / Paradas de prueba para funciones avanzadas
            res140_1 : Bool;
            res140_2 : Bool;
            res140_3 : Bool;
            res140_4 : Bool;
            CloseBrake : Bool;   // Interne Bremse schließen / Close internal Brake / Cerrar freno interno
            res140_6 : Bool;
            res140_7 : Bool;
            res141 : Byte;
         END_STRUCT;
         CW3 : Struct
            res142 : Byte;
            SelectionSBT : Bool;   // Auswahl: sicherer Bremstest / Selection: safe brake test / Selección: test de frenado seguro
            BT_Start : Bool;   // Start: Bremstest / Start: brake test / Inicio: test de frenado
            Brake_1_2 : Bool;   // Bremstest mit Bremse 1 oder 2 / Brake test with brake 1 or 2 / Test de frenado con freno 1 o 2
            DirOfROT : Bool;   // Drehrichtung / Direction of rotation / Sentido de giro
            Testseq_1_2 : Bool;   // Testsequenz 1 oder 2 / Test sequence 1 or 2 / Secuencia de test 1 o 2
            BrakeClosed : Bool;   // Rückmeldung externe Bremse / Feedback external brake / Respuesta freno externo
            res143_6 : Bool;
            res143_7 : Bool;
         END_STRUCT;
      END_STRUCT;
      res144_163 : Array[144..163] of Byte;
      SIC : Struct   // Antrieb zu PLC (SIC) / Drive to PLC (SIC) / Accionamiento a PLC (SIC)
         SW1 : Struct
            SLA_Sel : Bool;   // Sicher begrenzte Beschleunigung ausgewählt / Safely Limited Acceleration selected / Aceleración limitada con seguridad seleccionada
            SLS_LimBit0_Sel : Bool;   // Sicher begrenzte Geschwindigkeit: Grenze Bit0 ausgewählt / Safely-Limited Speed: limit Bit0 selected / Velocidad limitada con seguridad: límite bit 0 seleccionado
            SLS_LimBit1_Sel : Bool;   // Sicher begrenzte Geschwindigkeit: Grenze Bit1 ausgewählt / Safely-Limited Speed: limit Bit1 selected / Velocidad limitada con seguridad: límite bit 1 seleccionado
            res164_3 : Bool;
            res164_4 : Bool;
            res164_5 : Bool;
            ESR_Req : Bool;   // Erweiterter Stopp und Rückzug angefordert / Extended Stop and Retract requested / Parada ampliada y retirada solicitadas
            SF_Message_Act : Bool;   // Sicherheitsfehler aktiv / Safety error active / Error de seguridad activo
            STO_Act : Bool;   // Sicheres Drehmoment Aus: aktiv / Safe torque off: active / Desconexión segura de par: activa
            SS1_Act : Bool;   // Sicherer Stopp1: aktiv / Safe Stop1: active / Parada segura 1: activa
            SS2_Act : Bool;   // Sicherer Stopp2: aktiv / Safe Stop2: active / Parada segura 2: activa
            SOS_Act : Bool;   // Sicherer Betriebsstopp: aktiv / Safe Operating Stop: active / Parada de servicio segura: activa
            SLS_Act : Bool;   // Sicher begrenzte Geschwindigkeit: aktiv / Safely-Limited Speed: active / Velocidad limitada con seguridad: activa
            SOS_Sel : Bool;   // Sicherer Betriebsstopp: ausgewählt / Safe Operating Stop: selected / Parada de servicio segura: seleccionada
            SLS_Sel : Bool;   // Sicher begrenzte Geschwindigkeit: ausgewählt / Safely-Limited Speed: selected / Velocidad limitada con seguridad: seleccionada
            InternalEvent : Bool;   // Sicherheitsfehler mit Anschlag A aktiv / Safety error with Stop A active / Error de seguridad con tope A activo
         END_STRUCT;
         SW2 : Struct
            SDI_P_Sel : Bool;   // Sichere Richtung positiv: ausgewählt / Safe direction positive: selected / Sentido seguro positivo: seleccionado
            SDI_N_Sel : Bool;   // Sichere Richtung negativ: ausgewählt / Safe direction negative: selected / Sentido seguro negativo: seleccionado
            res166_2 : Bool;
            res166_3 : Bool;
            TestStopAct : Bool;   // Test-Stopp aktiv / Test stop active / Parada de prueba activa
            TestStopReq : Bool;   // Test-Stopp angefordert / Test stop requested / Parada de prueba solicitada
            res166_6 : Bool;
            res166_7 : Bool;
            res167_0 : Bool;
            res167_1 : Bool;
            res167_2 : Bool;
            res167_3 : Bool;
            SLP_LimBit0_Sel : Bool;   // Sicher begrenzte Position: Grenze Bit0 ausgewählt / Safely-Limited Position: limit Bit0 selected / Posición limitada con seguridad: límite bit 0 seleccionado
            res167_5 : Bool;
            res167_6 : Bool;
            SLP_Sel : Bool;   // Sicher begrenzte Position: ausgewählt / Safely-Limited Position: selected / Posición limitada con seguridad: seleccionada
         END_STRUCT;
         V_Limit_B : DInt;   // Solldrehzahlgrenze wirksam / Setpoint speed limit effective / Límite de consigna de velocidad efectivo
         SW3 : Struct
            res172_0 : Bool;
            res172_1 : Bool;
            res172_2 : Bool;
            SS2E_ACTIVE : Bool;   // SS2E aktiv / SS2E active / SS2E activo
            SS2ESR : Bool;   // SS2ESR aktiv / SS2ESR active / SS2ESR activo
            res172_5 : Bool;
            AcceptSLPAct : Bool;   // Abnahmetest sicher begrenzte Postion aktiv / Acceptance test Safely-Limited Position active / Prueba de recepción Posición limitada con seguridad activa
            AcceptTestSel : Bool;   // Abnahmetest ausgewählt / Acceptance test selected / Prueba de recepción seleccionada
            SBT_Sel : Bool;   // Sicherheitsbremstests: ausgewählt / Safety break test: selected / Test de frenado de seguridad: seleccionado
            SetpSettingDrive : Bool;   // Sollwerteingang ist beim SBT im Antrieb / Setpoint input is in the drive during the SBT / Entrada de consigna en el accionamiento durante SBT
            Brake_1_2 : Bool;   // Test mit Bremse 1 oder 2 / Test with brake 1 or 2 / Test con freno 1 o 2
            BT_Act : Bool;   // Bremstest: aktiv / Brake test: active / Test de frenado: activo
            BT_OK : Bool;   // Bremstest: OK / Brake test: OK / Test de frenado: OK
            BT_Finished : Bool;   // Bremstest: beendet / Brake test: finished / Test de frenado: finalizado
            BrakeReq : Bool;   // Externe Bremse schließen angefordert / External brake close requested / Solicitud cierre freno externo
            SignLoadTorque : Bool;   // Vorzeichen Lastmoment is negativ / Sign of load torque is negative / Signo de par de carga es negativo
         END_STRUCT;
      END_STRUCT;
      res174_187 : Array[174..187] of Byte;
      CW7 : Struct
         ReservedBit08 : Bool;
         ReservedBit09 : Bool;
         ReservedBit10 : Bool;
         ReservedBit11 : Bool;
         ReservedBit12 : Bool;
         ReservedBit13 : Bool;
         ReservedBit14 : Bool;
         ReservedBit15 : Bool;
         A_DisablePowerReduction : Bool;   // DYNEGMA: Leistungsreduktion deaktivieren / DYNEGMA: disable power reduction / DYNEGMA: desactivar reducción de potencia
         A_DisableCurrReduction : Bool;   // Motorübertemperatur: Stromreduktion deaktivieren / Motor overtemperature: disable current reduction / Exceso de temperatura en motor: desactivar reducción de corriente
         ReservedBit02 : Bool;
         ReservedBit03 : Bool;
         ReservedBit04 : Bool;
         ReservedBit05 : Bool;
         ReservedBit06 : Bool;
         ReservedBit07 : Bool;
      END_STRUCT;
      SW7 : Struct
         E_EncMaintenanceRequired : Bool;   // Geber-Instandhaltung erforderlich / Encoder maintenance required / Mantenimiento de encóder solicitado
         ReservedBit09 : Bool;
         ReservedBit10 : Bool;
         ReservedBit11 : Bool;
         ReservedBit12 : Bool;
         ReservedBit13 : Bool;
         ReservedBit14 : Bool;
         ReservedBit15 : Bool;
         E_TorqueLimited : Bool;   // DYNEGMA: Drehmoment begrenzt / DYNEGMA: torque limited / DYNEGMA: par limitado
         E_CurrReductionActive : Bool;   // Motorübertemperatur: Stromreduktion aktiv / Motor overtemperature: current reduction active / Exceso de temperatura en motor: reducción de corriente activa
         E_MotorTempModelAlarm : Bool;   // Motorübertemperatur: Alarm Motortemperaturmodell aktiv / Motor overtemperature: motor temperature model alarm active / Exceso de temperatura en motor: alarma modelo de temperatura del motor activa
         E_PolePosIdentPassed : Bool;   // Pollageidentifikation mit Geber erfolgreich durchgeführt / Pole position identification with encoder successfully carried out / Identificación de la posición polar con encóder realizada correctamente
         ReservedBit04 : Bool;
         ReservedBit05 : Bool;
         E_AndConditionFulfilled : Bool;   // Logische Verknüpfung UND: Bedingung erfüllt / AND logic operation: condition fulfilled / Operación lógica Y: condición cumplida
         E_OrConditionFulfilled : Bool;   // Logische Verknüpfung ODER: Bedingung erfüllt / OR logic operation: condition fulfilled / Operación lógica O: condición cumplida
      END_STRUCT;
   END_STRUCT;
END_TYPE

